// TwinCAT 3 PLC project Internship
// ProgramVersion: 3.1.4026.20
// libraries:
//   Tc2_Standard, * (Beckhoff Automation GmbH)
//   Tc2_System, * (Beckhoff Automation GmbH)
//   Tc3_Module, * (Beckhoff Automation GmbH)
// project tree:
//   Control/ FB_ControlSignal.TcPOU, FB_FeedForward.TcPOU, FB_FeedForward_NonLinear.TcPOU, FB_KvFF.TcPOU, FB_NaiveFF.TcPOU, FB_PID.TcPOU (not stored), FB_PressureFeedback.TcPOU, FB_Running.TcPOU (not stored), G_Mode.TcGVL (not stored)
//   Filtering/ FB_Filtering.TcPOU (not stored), G_Filtered.TcGVL (not stored)
//   GVL/ E_Mode.TcDUT (not stored), E_Motion.TcDUT, G_Enables.TcGVL, G_FilterConstants.TcGVL (not stored), G_OPC.TcGVL, G_Parameter.TcGVL
//   Inputs/Function Blocks/ FB_JoystickInputScaling.TcPOU, FB_Normalize.TcPOU (not stored), FB_PositionInputScaling.TcPOU
//   Inputs/ G_Inputs.TcGVL
//   MotionRef/ FB_AutoClock.TcPOU (not stored), FB_Home.TcPOU, FB_InitialPos.TcPOU (not stored), FB_MotionRef.TcPOU, FB_RunClock.TcPOU (not stored)
//   Outputs/ FB_ValveOutput.TcPOU (not stored), G_Output.TcGVL (not stored)
//   / PlcTask.TcTTO (not stored)
//   Programs/ MAIN.TcPOU (not stored), P_ControlBlock.TcPOU, P_FeedForward.TcPOU, P_Filtering.TcPOU (not stored), P_Inputs.TcPOU, P_Modes.TcPOU (not stored), P_Output.TcPOU, P_PID.TcPOU (not stored), P_RunClock.TcPOU (not stored)
//   XML/ FB_Derivator.TcPOU (not stored), G_Init.TcGVL (not stored), FB_Integrator.TcPOU (not stored)
// real-time tasks:
//   TASK PlcTask: cycle T#1ms, priority 20, ADS port 350
// I/O:
//   DEVICE Device 3 (EtherCAT), AmsNetId 192.168.0.204.4.1
//     RIO (EK1100) [EK1100 EtherCAT Coupler (2A E-Bus)]
//       DI (EL1008) [EL1008 8Ch. Dig. Input 24V, 3ms]
//       DO (EL2008) [EL2008 8Ch. Dig. Output 24V, 0.5A]
//       AI1 (EL3068) [EL3068 8Ch. Ana. Input 0-10V]
//       AI2 (EL3068) [EL3068 8Ch. Ana. Input 0-10V]
//       AI3 (EL3174) [EL3174 4Ch. Ana. Input +/-10V Diff., +/-20mA SingleEnded, 16 Bit]
//       AO (EL4104) [EL4104 4Ch. Ana. Output 0-10V, 16bit]
//       End Cap (EL9011) [EL9011 End Terminal]
// variable links:
//   Internship/Internship Instance <-> Device 3 (EtherCAT)/RIO (EK1100)/AI1 (EL3068)
//     PlcTask Inputs/G_Inputs.nRawJoystick <-> AI Standard Channel 2/Value
//     PlcTask Inputs/G_Inputs.nRawPistonPosition <-> AI Standard Channel 3/Value
//     PlcTask Inputs/G_Inputs.nRawSpoolPosition <-> AI Standard Channel 4/Value
//   Internship/Internship Instance <-> Device 3 (EtherCAT)/RIO (EK1100)/AI2 (EL3068)
//     PlcTask Inputs/G_Inputs.nRawPa <-> AI Standard Channel 4/Value
//     PlcTask Inputs/G_Inputs.nRawPaLower <-> AI Standard Channel 5/Value
//     PlcTask Inputs/G_Inputs.nRawPb <-> AI Standard Channel 6/Value
//     PlcTask Inputs/G_Inputs.nRawPs <-> AI Standard Channel 1/Value
//   Internship/Internship Instance <-> Device 3 (EtherCAT)/RIO (EK1100)/AI3 (EL3174)
//     PlcTask Inputs/G_Inputs.nRawFlowSensor <-> AI Standard Channel 1/Value
//   Internship/Internship Instance <-> Device 3 (EtherCAT)/RIO (EK1100)/AO (EL4104)
//     PlcTask Outputs/G_Output.nValveOutput <-> AO Output Channel 1/Analog output
//   Internship/Internship Instance <-> Device 3 (EtherCAT)/RIO (EK1100)/DI (EL1008)
//     PlcTask Inputs/G_Inputs.bAuto <-> Channel 1/Input
//     PlcTask Inputs/G_Inputs.bManual <-> Channel 2/Input
//     PlcTask Inputs/G_Inputs.bStartButton <-> Channel 3/Input
//     PlcTask Inputs/G_Inputs.bStopButton <-> Channel 4/Input
//   Internship/Internship Instance <-> Device 3 (EtherCAT)/RIO (EK1100)/DO (EL2008)
//     PlcTask Outputs/G_Output.bGreenLight <-> Channel 1/Output
//     PlcTask Outputs/G_Output.bRedLight <-> Channel 2/Output
//     PlcTask Outputs/G_Output.bRunning <-> Channel 3/Output

// ---- GVL/E_Motion.TcDUT
{attribute 'qualified_only'}
{attribute 'strict'}
{attribute 'to_string'}
TYPE E_Motion :
(
	Sine,
	Ramp
);
END_TYPE

// ---- GVL/G_Enables.TcGVL
{attribute 'qualified_only'}
VAR_GLOBAL
	
	// Control Enables
	bEnablePID 		: BOOL; // Enable PID Control
	bEnableFF 		: BOOL; // Enable FeedForward	
	bEnablePFB		: BOOL; // Enable Pressure Feedback
	bEnableU 		: BOOL; // Enable Signal to Valve

	bCharTesting	: BOOL; // Enable Characteristic testing
	bMove2Home		: BOOL; // Enable Home-function
	
	// No Function
	bEnableComp 	: BOOL; // Driving with Compensator
	

	// Enumerators
	nModeSelect		: E_Motion; // Motion Reference
	
END_VAR

// ---- GVL/G_OPC.TcGVL
{attribute 'qualified_only'}
VAR_GLOBAL
	
	// Unfiltered Pressures
	fPa 				: LREAL; // [bar], Pressure A 
	fPb 				: LREAL; // [bar], Pressure B 
	fPs 				: LREAL; // [bar], Pressure S 
	fPaLower 			: LREAL; // [bar], Pressure A inbetween DCV and CBV 
	
	// Filtered Pressures
	fPaFiltered 		: LREAL; // [bar], Pressure A Filtered 
	fPbFiltered 		: LREAL; // [bar], Pressure B Filtered
	fPsFiltered 		: LREAL; // [bar], Pressure S Filtered
	fPaLowerFiltered 	: LREAL; // [bar], Pressure A inbetween DCV and CBV Filtered
	
	fSpoolPosition 		: LREAL; // [-1..1], Spool position 
	fPistonPosition 	: LREAL; // [m], Piston position
	fPistonPosMeasured 	: LREAL; // [m], Measured piston position
	fJoystick 			: LREAL; // [-1..1], Joystick signal
	fFlow 				: LREAL; // [l/min], Flow rod side 
	fFlowCalc 			: LREAL; // [l/min], Calculated flow
	
	fXRef 				: LREAL; // [m], Position reference [m]
	fXDotRef 			: LREAL; // [m/s], Velocity reference [m/s]
	fFlowRef 			: LREAL; // [l/min], Flow reference calculated form fXDotRef
	
	fFFFlow				: LREAL; // [l/min], Flow form feed forward
	fKv					: LREAL;

	fWantedSpoolPos 	: LREAL; // [-1..1], Where spool is wanted to be
	fUpfbGrad 			: LREAL; // Pressure feedback gradient
	fPxGrad 			: LREAL; // Pressure gradient
	fUTest 				: LREAL; // [-1..1], Signal to Valve with pfb
	fTime 				: LREAL; // [s], Time
	fError 				: LREAL; // [m], Error
	
	
	fSignalPID 			: LREAL; // PID signal value
	fFF 				: LREAL; // FF signal Value
	fUpfb 				: LREAL; // Pressure feedback signal
	fU 					: LREAL; // [-1..1], Signal for spool to be where it is wanted


END_VAR

// ---- GVL/G_Parameter.TcGVL
{attribute 'qualified_only'}
VAR_GLOBAL
	// Motion Ref
	// Sine Parameters
	fAmplitude 		: LREAL := 0.15;
	fMean 			: LREAL := 0.2;
	fFrequency 		: LREAL := 0.05;
	
	
	// Valve Values
	// Flow
	fQMaxDown 		: LREAL := 10.0; // [L/min]
	fQMaxUp 		: LREAL := 10.0; // [L/min]	
	
	// Area
	fAreaUp 		: LREAL := 33.100/1E4; //[m^2]
	fAreaDown 		: LREAL := 23.560/1E4; //[m^2]
	
	// Deadband
	fDeadUp 		: LREAL := 0.23;
	fDeadDown 		: LREAL := 0.215;
	
	fMaxSpeed 		: LREAL := 0.01; // [m/s] 
	fDeltaP0 		: LREAL := 8.0; // [Bar]
	
	// Deadband test
	fConst 			: LREAL := 0.0; // [-1, 1]

	fCycleTime 		: LREAL := 0.001; // Time Step [s]
	fQConst 		: LREAL := 15;
	fPistonStroke 	: LREAL := 0.5;
	
	// PID-constants
	Kp 				: LREAL := 14.0; 	// P
	Ki 				: LREAL := 0.0;		// I
	Kd 				: LREAL := 0.0;		// D
	
	// Pressure feedback constants
	Kf				: LREAL := 2E-4;
	TauF			: LREAL := 0.1; // [0.05 .. 0.1]
	PFBstate		: INT 	:= 2; // 0:Switching, 1: Pa-phi*Pb, 2: Pb
	FFMode			: INT 	:= 1; // 0: Bachelor FF, 1: Kv FF, 2: Naive FF




END_VAR

// ---- Inputs/G_Inputs.TcGVL
{attribute 'qualified_only'}
VAR_GLOBAL
	// Mode Selector
	bManual 			AT %I* : BOOL;
	bAuto	 			AT %I* : BOOL;
	bStartButton		AT %I* : BOOL;
	bStopButton			AT %I* : BOOL;
	
	// Raw Pressure Values
	nRawPa 				AT %I*	: INT;
	nRawPb				AT %I*	: INT;
	nRawPs				AT %I*	: INT;
	nRawPaLower			AT %I* 	: INT;
	
	// Raw Position Values
	nRawPistonPosition 	AT %I*	: INT;
	nRawJoystick		AT %I*	: INT;
	nRawFlowSensor		AT %I*	: INT;
	nRawSpoolPosition	AT %I*	: INT;
END_VAR

// ---- Control/FB_ControlSignal.TcPOU
FUNCTION_BLOCK FB_ControlSignal
VAR_INPUT
	fFF 			: LREAL;
	fPID			: LREAL;
	fPFB			: LREAL;
	
	fDeadBandUp		: LREAL;
	fDeadBandDown	: LREAL;
	
	nFFState		: INT;

	bPID			: BOOL;
	bFF				: BOOL;
	bPFB			: BOOL;
	bU				: BOOL;
	bValve			: BOOL;
END_VAR
VAR_OUTPUT
	fU				: LREAL;
	fUAdj			: LREAL;
END_VAR
VAR
	FF				: LREAL;
	PID				: LREAL;
	PFB				: LREAL;
END_VAR


FF := fFF  * TO_INT(bFF);

PID := fPID * TO_INT(bPID);

PFB := fPFB * TO_INT(bPFB);

fUAdj := (FF+PID-PFB)*TO_INT(bValve);

IF FF = 0.0 THEN
	fU := 0.0;
ELSE
	CASE nFFState OF
		0: 
			IF (fUAdj > 0.0) THEN
				fU := fUAdj + fDeadBandUp;
			ELSIF (fUAdj < 0.0) THEN
				fU := fUAdj - fDeadBandDown;
			ELSE
				fU := 0.0;
			END_IF
			
		ELSE // FF States that use this: 1, 2
			IF (fUAdj > 0.0) THEN
				fU := fUAdj;
			ELSIF (fUAdj < 0.0) THEN
				fU := fUAdj;
			ELSE
				fU := 0.0;
			END_IF

		
	END_CASE
	
END_IF
IF fU < -1.0 THEN
	fU := -1.0;
ELSIF fU > 1.0 THEN
	fU := 1.0;
ELSE
	fU := fU;
END_IF

END_FUNCTION_BLOCK

// ---- Control/FB_FeedForward.TcPOU
FUNCTION_BLOCK FB_FeedForward
VAR_INPUT
	fXDotRef 		: LREAL; // Velocity Reference [m/s]
	fMaxFlowUp 		: LREAL; // Needs to be positive (22)
	fMaxFlowDown 	: LREAL; // Needs to be positive (15)
	fDeadUp			: LREAL; // Needs to be positive (0.155)
	fDeadDown 		: LREAL; // Needs to be positive (0.18)

	fPs 			: LREAL; // [Bar]
	fPa 			: LREAL; // [Bar]
	fPb 			: LREAL; // [Bar]
	fDeltaP0		: LREAL; // [Bar]
	fAreaUp			: LREAL; // [mm^2]
	fAreaDown		: LREAL; // [mm^2]

END_VAR
VAR_OUTPUT
	fUFF 			: LREAL;
	fFlow			: LREAL; 	// Wanted Flow
	fFlowLM			: LREAL;	// Flow [L/min]
END_VAR
VAR

	fDeltaP_Norm	: LREAL; 	// Pressure Drop with Compansator
	
	fDeltaP			: LREAL; 	// Pressure Drop
	fDeltaP_Ref		: LREAL; 	// Referance Pressure Drop
	fFlowRef		: LREAL; 	// Refereance Flow
	
	fUFFTemp		: LREAL;	// Temp Signal Out
END_VAR


fDeltaP_Norm	:= fDeltaP0 * 100000.0;

IF fXDotRef > 0.0 THEN
	
	fFlow := fXDotRef * fAreaUp;
	fFlowLM := -fFlow * 60000;
	fDeltaP := (fPs - fPa) * 100000.0;
	IF fDeltaP < 100 THEN
		fDeltaP := 100;
	ELSE
		fDeltaP := fDeltaP;
	END_IF
	fDeltaP_Ref := ABS(fDeltaP_Norm/ (fDeltaP));
	fFlowRef := (fFlow * SQRT(fDeltaP_Ref)) * 60000.0;
	fUFFTemp := fFlowRef/fMaxFlowUp;
	fUFFTemp := -fUFFTemp * (1.0-fDeadUp);
	
ELSIF fXDotRef < 0.0 THEN
	
	fFlow := fXDotRef * fAreaDown;
	fFlowLM := -fFlow * 60000;
	fDeltaP := (fPs - fPb) * 100000.0;
	IF fDeltaP < 100 THEN
		fDeltaP := 100;
	ELSE
		fDeltaP := fDeltaP;
	END_IF
	fDeltaP_Ref := ABS(fDeltaP_Norm/(fDeltaP));
	fFlowRef := (fFlow * SQRT(fDeltaP_Ref)) * 60000.0;
	fUFFTemp := fFlowRef/fMaxFlowDown; 
	fUFFTemp := -fUFFTemp*(1.0-fDeadDown);
	
ELSE
	
	fUFFTemp := 0.0;		

END_IF

IF fUFFTemp > 1.0 THEN
	fUFF := 1.0;
ELSIF fUFFTemp < -1.0 THEN
	fUFF := -1.0;
ELSE
	fUFF := fUFFTemp;
END_IF

END_FUNCTION_BLOCK

// ---- Control/FB_FeedForward_NonLinear.TcPOU
FUNCTION_BLOCK FB_FeedForward_NonLinear
VAR_INPUT
	fXDotRef 		: LREAL; // Velocity Reference [m/s]
	fMaxFlowUp 		: LREAL; // Needs to be positive (22)
	fMaxFlowDown 	: LREAL; // Needs to be positive (15)
	fDeadUp			: LREAL; // Needs to be positive (0.155)
	fDeadDown 		: LREAL; // Needs to be positive (0.18)

	fPs 			: LREAL; // [Bar]
	fPa 			: LREAL; // [Bar]
	fPb 			: LREAL; // [Bar]
	fDeltaP0		: LREAL; // [Bar]
	fAreaUp			: LREAL; // [mm^2]
	fAreaDown		: LREAL; // [mm^2]

END_VAR
VAR_OUTPUT
	fUFF 			: LREAL;
	fFlow			: LREAL; 	// Wanted Flow
	fFlowLM			: LREAL;	// Flow [L/min]
END_VAR
VAR

	fDeltaP_Norm	: LREAL; 	// Pressure Drop with Compansator
	
	fDeltaP			: LREAL; 	// Pressure Drop
	fDeltaP_Ref		: LREAL; 	// Referance Pressure Drop
	fFlowRef		: LREAL; 	// Refereance Flow
	
	fUFFTemp		: LREAL;	// Temp Signal Out
END_VAR


fDeltaP_Norm	:= fDeltaP0 * 100000.0;

IF fXDotRef > 0.0 THEN
	
	fFlow := fXDotRef * fAreaUp;
	fFlowLM := -fFlow * 60000;
	fDeltaP := (fPs - fPa) * 100000.0;
	IF fDeltaP < 100 THEN
		fDeltaP := 100;
	ELSE
		fDeltaP := fDeltaP;
	END_IF
	fDeltaP_Ref := ABS(fDeltaP_Norm/ (fDeltaP));
	fFlowRef := (fFlow * SQRT(fDeltaP_Ref)) * 60000.0;
	fUFFTemp := fFlowRef/fMaxFlowUp;
	fUFFTemp := -fUFFTemp * (1.0-fDeadUp);
	
ELSIF fXDotRef < 0.0 THEN
	
	fFlow := fXDotRef * fAreaDown;
	fFlowLM := -fFlow * 60000;
	fDeltaP := (fPs - fPb) * 100000.0;
	IF fDeltaP < 100 THEN
		fDeltaP := 100;
	ELSE
		fDeltaP := fDeltaP;
	END_IF
	fDeltaP_Ref := ABS(fDeltaP_Norm/(fDeltaP));
	fFlowRef := (fFlow * SQRT(fDeltaP_Ref)) * 60000.0;
	fUFFTemp := fFlowRef/fMaxFlowDown; 
	fUFFTemp := -fUFFTemp*(1.0-fDeadDown);
	
ELSE
	
	fUFFTemp := 0.0;		

END_IF

IF fUFFTemp > 1.0 THEN
	fUFF := 1.0;
ELSIF fUFFTemp < -1.0 THEN
	fUFF := -1.0;
ELSE
	fUFF := fUFFTemp;
END_IF

END_FUNCTION_BLOCK

// ---- Control/FB_KvFF.TcPOU
FUNCTION_BLOCK FB_KvFF
VAR_INPUT
	fPs 		: LREAL; // [bar]
	fPa 		: LREAL; // [bar]
	fPb 		: LREAL; // [bar]
	
	fXDotRef 	: LREAL; // [m/s]
END_VAR
VAR_OUTPUT
	fFFTemp		: LREAL; // [-1..1], Wanted spool position, u
	fFF 		: LREAL; // [-1..1], Spool signal for position, ~u
	fFlow 		: LREAL; // [l/min]
	fKv 		: LREAL; // [l/min / bar^0.5]
END_VAR
VAR
	fDeltaP		: LREAL; // [bar]
END_VAR




IF fXDotRef > 0.0 THEN
	IF fKv >= 0.1 THEN
		fFFTemp := -0.013*EXPT(fKv,5) + 0.1355*EXPT(fKv,4) - 0.5012*EXPT(fKv,3) + 0.7175*EXPT(fKv,2) - 0.0278 * fKv + 0.2684;
	ELSIF fKv < 0.1 THEN
		fFFTemp := 0.2325 + 0.0398 * fKv/0.1;
	ELSE 
		fFFTemp := G_Parameter.fDeadUp;
	END_IF
	fFlow := fXDotRef * G_Parameter.fAreaUp * 6E4;
	fDeltaP := fPs - fPa;
	
	fFF := -(fFFTemp + 0.0151)/1.1224;
ELSIF fXDotRef < 0.0 THEN
	IF fKv >= 0.1 THEN
		fFFTemp := 0.0054*EXPT(fKv,6) - 0.0733*EXPT(fKv,5) + 0.3796*EXPT(fKv,4) - 0.9356*EXPT(fKv,3) + 1.0359*EXPT(fKv,2) - 0.1046 * fKv + 0.2381;
	ELSIF fKv < 0.1 THEN
		fFFTemp := 0.2175 + 0.0196 * fKv/0.1;
	ELSE 
		fFFTemp := G_Parameter.fDeadDown;
	END_IF
	fFlow := fXDotRef * G_Parameter.fAreaDown * 6E4;
	fDeltaP := fPs - fPb;
	fFF := (fFFTemp + 0.0398)/1.1079;
ELSE
	fFlow := 0.0;
	fFFTemp := 0.0;
	fFF := 0.0;
END_IF

IF fDeltaP <= 0.0 THEN
	fKv := 4.0;
ELSE
	fKv := ABS(fFlow)/SQRT(fDeltaP);
END_IF

END_FUNCTION_BLOCK

// ---- Control/FB_NaiveFF.TcPOU
FUNCTION_BLOCK FB_NaiveFF
VAR_INPUT
	fPs 		: LREAL; // [bar]
	fPa 		: LREAL; // [bar]
	fPb 		: LREAL; // [bar]
	
	fXDotRef 	: LREAL; // [m/s]
END_VAR
VAR_OUTPUT

	fFF 		: LREAL; // [-1..1], Spool signal for position, u
	fFlow 		: LREAL; // [l/min]
	fKv 		: LREAL; // [l/min / bar^0.5]
END_VAR
VAR
	fDeltaP		: LREAL; // [bar]
END_VAR




IF fXDotRef > 0.0 THEN
	fFlow := fXDotRef * G_Parameter.fAreaUp * 6E4;
	fDeltaP := fPs - fPa;
	
	fFF := -(0.2143 + 0.7857 * fKv/3.7796);
ELSIF fXDotRef < 0.0 THEN
	fFlow := fXDotRef * G_Parameter.fAreaDown * 6E4;
	fDeltaP := fPs - fPb;
	
	fFF := (0.2143 + 0.7857 * fKv/3.7796);
ELSE
	fFlow := 0.0;
	fFF := 0.0;
END_IF

IF fDeltaP <= 0.0 THEN
	fKv := 4.0;
ELSE
	fKv := ABS(fFlow)/SQRT(fDeltaP);
END_IF

END_FUNCTION_BLOCK

// ---- Control/FB_PressureFeedback.TcPOU
FUNCTION_BLOCK FB_PressureFeedback
VAR_INPUT
	fKf			: LREAL;
	fTauF		: LREAL; // [s]	
	state		: INT;
END_VAR
VAR_OUTPUT
	fUpfb 		: LREAL;
	fUpfbGrad	: LREAL;
	fPxGrad		: LREAL; // [Bar]
END_VAR
VAR
	fDt			: LREAL := 0.001; // [s]
	fPx			: LREAL := 0.0; // [Bar]
	fPxOld		: LREAL; // [Bar]
	fARatio		: LREAL;
END_VAR


CASE state OF
	0: // Altering input for Px
		IF G_OPC.fU < 0.0 THEN
			fPx := G_OPC.fPa;
		ELSIF G_OPC.fU > 0.0 THEN
			fPx := G_OPC.fPb;
		ELSE
			fPx := 0.0;
		END_IF
	1:	// Px = Pa - phi * Pb
		fARatio := G_Parameter.fAreaDown/G_Parameter.fAreaUp;
		fPx := G_OPC.fPa - fARatio * G_OPC.fPb;
	2:	// Px = Pb
		fPx := G_OPC.fPb;
END_CASE

fPxGrad := (fPx - fPxOld)/fDt;
fUpfbGrad :=  (fKf * fPxGrad - fUpfb)/fTauF;
fUpfb := fUpfb + fUpfbGrad * fDt;

fPxOld := fPx;

END_FUNCTION_BLOCK

// ---- Inputs/Function Blocks/FB_JoystickInputScaling.TcPOU
FUNCTION_BLOCK FB_JoystickInputScaling
VAR_INPUT
	bEnable 				: BOOL;
	nRawInput 				: INT;
	fMaxValue 				: LREAL;
	fMaxInputValue			: LREAL;
	fMinInputValue 			: LREAL;
	fNeutralInputValue  	: LREAL;
	fNeutralDeadband		: LREAL;
END_VAR
VAR_OUTPUT
	fOutput : LREAL;
END_VAR
VAR
	fRawInput : LREAL;
	fTempInput : LREAL;
	fTempOutput : LREAL;

	fMaxOutputValue  		: LREAL := 1.0;
	fMinOutputValue  		: LREAL := -1.0;
	fNeutralOutputValue  	: LREAL := 0.0;
END_VAR

fRawInput := INT_TO_LREAL(nRawInput);

fTempInput := fRawInput - fNeutralInputValue;

IF fTempInput > fNeutralDeadband THEN
	fTempOutput := fTempInput/(fMaxInputValue - fNeutralInputValue);
ELSIF fTempInput < -fNeutralDeadband THEN	
	fTempOutput := fTempInput/(fNeutralInputValue - fMinInputValue);
ELSE
	fTempOutput := 0.0;
END_IF

IF NOT(bEnable) THEN
	fOutput := 0.0;
ELSE
	fOutput := LIMIT(fMinOutputValue * fMaxValue, fTempOutput * fMaxValue, fMaxOutputValue* fMaxValue);
END_IF

END_FUNCTION_BLOCK

// ---- Inputs/Function Blocks/FB_PositionInputScaling.TcPOU
FUNCTION_BLOCK FB_PositionInputScaling
VAR_INPUT
	nRawInput 				: INT;
	fMaxInputValue 			: LREAL;
	fMinInputValue			: LREAL;
	fMaxOutputValue  		: LREAL;
	fMinOutputValue  		: LREAL;	
END_VAR
VAR_OUTPUT
	fOutput : LREAL;
	fActual : LREAL;
END_VAR
VAR
	fRawInput : LREAL;
	fNormalizedInput: LREAL;
	fTempOut : LREAL;
END_VAR

fRawInput := INT_TO_LREAL(nRawInput);

fNormalizedInput := (fRawInput - fMinInputValue) / (fMaxInputValue - fMinInputValue);
fTempOut := fMinOutputValue + fNormalizedInput*(fMaxOutputValue - fMinOutputValue);

fOutput := LIMIT(fMinOutputValue, fTempOut, fMaxOutputValue);
fActual := LIMIT(fMinOutputValue, fTempOut - 0.0006 - 0.0109*fTempOut + 0.5855*EXPT(fTempOut,2) - 1.1291*EXPT(fTempOut,3), fMaxOutputValue);

END_FUNCTION_BLOCK

// ---- MotionRef/FB_Home.TcPOU
FUNCTION_BLOCK FB_Home
VAR_INPUT
	bGoHome : BOOL;
	fCurrentPos : LREAL; // [m]
	fTolerance : LREAL; // [m]
	fMoveTime : LREAL; // [s]
	fHomePos : LREAL; // [m]
	fMoveTimer : LREAL; // [s]
END_VAR
VAR_OUTPUT
	fXRef : LREAL; // [m]
	fXDotRef : LREAL; // [m/s]
END_VAR
VAR
	
END_VAR




IF bGoHome AND ABS(fHomePos-fCurrentPos)>fTolerance THEN
	fXDotRef := (fHomePos-fCurrentPos)/fMoveTime;
	fXRef := fCurrentPos + fXDotRef * fMoveTimer;
	IF	ABS(fHomePos-fCurrentPos)<=fTolerance THEN
		bGoHome := FALSE;
		fXDotRef := 0.0;
		fXRef := fCurrentPos;
	END_IF
ELSE
	fXDotRef := 0.0;
	fXRef := fCurrentPos;
END_IF

END_FUNCTION_BLOCK

// ---- MotionRef/FB_MotionRef.TcPOU
FUNCTION_BLOCK FB_MotionRef
VAR_INPUT
	fAmplitude : LREAL;
	fFrequency : LREAL;
	fInitialPos : LREAL;
	fCurrentPos : LREAL;
	nMotionMode : INT;
	fMotionTimer 	: LREAL;           // For selve rampen
END_VAR
VAR_OUTPUT
	fXDotRef : LREAL;
	fXRef : LREAL;
	fWantedFlow : LREAL;
END_VAR
VAR
	fPI : LREAL := 3.1415;
	fMean : LREAL;
	
	arrBounduary 	: ARRAY[0..1] OF LREAL := [G_Parameter.fPistonStroke * 0.1, G_Parameter.fPistonStroke * 0.9]; // Min, Max [m]
	fRampTime 	 	: LREAL := 15.0; // [s]
 	fTolerance   	: REAL := 0.005;  // ±5 mm
  	
END_VAR




CASE nMotionMode OF
	0:	// Sine
	
		fMean := fAmplitude + fInitialPos; 
		fXRef := fMean - fAmplitude * COS(2*fPI * fFrequency * fMotionTimer);
		fXDotRef := 2 * fPI *fFrequency * fAmplitude * SIN(2*fPI * fFrequency * fMotionTimer); 
		
	1:	// Ramp


		IF fMotionTimer <= fRampTime THEN
			fXDotRef := (arrBounduary[1] - arrBounduary[0]) / fRampTime;
			fXRef := arrBounduary[0] + fXDotRef * fMotionTimer;
		ELSIF fMotionTimer <= fRampTime * (4.0/3.0) THEN
			fXRef := arrBounduary[1];
			fXDotRef := 0.0;
		ELSIF fMotionTimer <= (2.0 + 1.0/3.0) * fRampTime AND fMotionTimer > fRampTime * (4.0/3.0) THEN
			fXDotRef := (arrBounduary[0] - arrBounduary[1]) / fRampTime;
			fXRef := arrBounduary[1] + fXDotRef * (fMotionTimer - (4.0/3.0) * fRampTime);
		ELSIF fMotionTimer > (2.0 + 1.0/3.0) * fRampTime THEN
			fXDotRef := 0.0;
			fXRef := arrBounduary[0];
		END_IF
END_CASE

IF fXDotRef > 0.0 THEN
	fWantedFlow := fXDotRef * G_Parameter.fAreaUp*6E4;
ELSIF fXDotRef < 0.0 THEN
	fWantedFlow := fXDotRef * G_Parameter.fAreaDown*6E4;
ELSE
	fWantedFlow := 0.0;
END_IF

END_FUNCTION_BLOCK

// ---- Programs/P_ControlBlock.TcPOU
PROGRAM P_ControlBlock
VAR
	fbAutoClock : FB_AutoClock;
	fbMotionRef : FB_MotionRef;
	fbControl : FB_ControlSignal;
	fbInitialPos : FB_InitialPos;
	nMode : E_Motion;
	fbPressureFB : FB_PressureFeedback;
	fbHome : FB_Home;
	StartTimer : TON;
END_VAR


fbControl(
	nFFState := G_Parameter.FFMode,	

	bFF := G_Enables.bEnableFF,
	bPID := G_Enables.bEnablePID,
	bPFB := G_Enables.bEnablePFB,
	bU := G_Enables.bEnableU,
	bValve := TRUE,
	
	fDeadBandUp := G_Parameter.fDeadUp,
	fDeadBandDown := G_Parameter.fDeadDown
);

fbPressureFB(
			fKf := G_Parameter.Kf,
			fTauF := G_Parameter.TauF,
			state := G_Parameter.PFBstate,
			
			fUpfb => G_OPC.fUpfb,
			fUpfbGrad => G_OPC.fUpfbGrad,
			fPxGrad => G_OPC.fPxGrad
		);

IF G_Mode.bAuto AND G_Mode.bRunning THEN

	fbInitialPos(
		bEnable := G_Inputs.bStartButton,
		fCurrentPos := G_OPC.fPistonPosition
	);
	
	fbAutoClock(
		fStart := StartTimer.Q,
		fRunning := G_Mode.bRunning,
		fCycle := G_Parameter.fCycleTime
	);
	
	IF G_Inputs.bStartButton THEN
		StartTimer(IN := TRUE, PT :=T#2S);
		fbMotionRef();
		IF StartTimer.Q THEN
			
			IF G_Enables.bMove2Home THEN 
				fbHome(
					bGoHome := G_Enables.bMove2Home,
					fCurrentPos := G_OPC.fPistonPosition,
					fHomePos := 0.05,
					fMoveTimer := fbAutoClock.fTime,
					fMoveTime := 10.0,
					fTolerance := 0.002,
					
					fXDotRef => G_OPC.fXDotRef,
					fXRef => G_OPC.fXRef
				);
			ELSE
			fbMotionRef(
				nMotionMode := G_Enables.nModeSelect,
				fMotionTimer := fbAutoClock.fTime,
				fAmplitude := G_Parameter.fAmplitude,
				fInitialPos := fbInitialPos.fInitialPos,
				fFrequency := G_Parameter.fFrequency,
				fCurrentPos := G_OPC.fPistonPosition,
				fXDotRef => G_OPC.fXDotRef,
				fXRef => G_OPC.fXRef,
				fWantedFlow => G_OPC.fFlowRef
			);
			END_IF
		ELSE 
			G_OPC.fXDotRef := 0.0;
			G_OPC.fXRef := G_OPC.fPistonPosition;
		END_IF
	ELSE 
		StartTimer(IN := FALSE);
		G_OPC.fXDotRef := 0.0;
		G_OPC.fXRef := G_OPC.fPistonPosition;
	END_IF
	
	
	G_OPC.fUTest := G_OPC.fU - G_OPC.fUpfb;
	
	fbControl(
		fFF := G_OPC.fFF,
		fPID := G_OPC.fSignalPID,
		fPFB := G_OPC.fUpfb,
		
		fU => G_OPC.fU
	);
		
		
	
	

ELSIF G_Mode.bManual AND G_Mode.bRunning THEN

	fbInitialPos(
		bEnable := G_Inputs.bStartButton,
		fCurrentPos := G_OPC.fPistonPosition
	);
	
	IF G_Enables.bCharTesting THEN
		IF G_OPC.fPistonPosition >= 0.9*0.5 OR G_OPC.fPistonPosition <= 0.1 * 0.5 THEN
			G_OPC.fU := 0.0;
		ELSE
			G_OPC.fU := G_Parameter.fConst - G_OPC.fUpfb * TO_INT(G_Enables.bEnablePFB);
		END_IF
	
	ELSE
		G_OPC.fU := G_OPC.fJoystick;
	END_IF
	
END_IF

END_PROGRAM

// ---- Programs/P_FeedForward.TcPOU
PROGRAM P_FeedForward
VAR
	fbFF 	: FB_FeedForward;
	fbKv 	: FB_KvFF;
	fbNaive	: FB_NaiveFF;
END_VAR

//fbKv(
//	fPa := G_OPC.fPa,
//	fPb := G_OPC.fPb,
//	fPs := G_OPC.fPs,
	
//	fXDotRef := G_OPC.fXDotRef,
	
//	fUTemp => G_OPC.fWantedSpoolPos,
//	fU => G_OPC.fU
//);

	
CASE G_Parameter.FFMode OF
	0:
		fbFF(
			fMaxFlowUp := G_Parameter.fQMaxUp,
			fMaxFlowDown := G_Parameter.fQMaxDown,
			fDeadUp := G_Parameter.fDeadUp,
			fDeadDown := G_Parameter.fDeadDown,
			fAreaUp := G_Parameter.fAreaUp,
			fAreaDown := G_Parameter.fAreaDown,
			
			fPs := G_OPC.fPs,
			fPa := G_OPC.fPa,
			fPb := G_OPC.fPb,
			fDeltaP0 := G_Parameter.fDeltaP0,
			
			fXDotRef := G_OPC.fXDotRef,		
	
			fUFF => G_OPC.fFF,
			fFlowLM => G_OPC.fFlowCalc
		);
		
	1:
		fbKv(
			fPa :=G_OPC.fPaLower,
			fPb := G_OPC.fPb,
			fPs := G_OPC.fPs,
			
			fXDotRef := G_OPC.fXDotRef,
			
			fFFTemp => G_OPC.fWantedSpoolPos,
			fFF => G_OPC.fFF,
			fFlow => G_OPC.fFFFlow,
			fKv => G_OPC.fKv
			
			
		);
	2:
		fbNaive(
			fPa :=G_OPC.fPaLower,
			fPb := G_OPC.fPb,
			fPs := G_OPC.fPs,
			
			fXDotRef := G_OPC.fXDotRef,
			
			fFF => G_OPC.fFF,
			fFlow => G_OPC.fFFFlow,
			fKv => G_OPC.fKv
		);
		

END_CASE

END_PROGRAM

// ---- Programs/P_Inputs.TcPOU
PROGRAM P_Inputs
VAR
	fbNormPa :  FB_Normalize;
	fbNormPb :  FB_Normalize;
	fbNormPs :  FB_Normalize;
	fbNormPaLower : FB_Normalize;
	
	fbNormPistonPosition : FB_PositionInputScaling;
	fbNormSpoolPosition : FB_JoystickInputScaling;
	fbJoystick : FB_JoystickInputScaling;
	fbFlow	: FB_JoystickInputScaling;

	fPa : LREAL;
	fPb : LREAL;
	fPs : LREAL;
	fPaLower : LREAL;
	
	fPistonPosition : LREAL;
END_VAR

fbNormPa(
	nRawInput := G_Inputs.nRawPa,
	fMaxValue := 400.0, 			// [Bar]
	fNormalizedInput => G_OPC.fPa
);

fbNormPb(
	nRawInput := G_Inputs.nRawPb,
	fMaxValue := 400.0, 			// [Bar]
	fNormalizedInput => G_OPC.fPb
);

fbNormPs(
	nRawInput := G_Inputs.nRawPs,
	fMaxValue := 400.0, 			// [Bar]
	fNormalizedInput => G_OPC.fPs
);

fbNormPistonPosition(
	nRawInput := G_Inputs.nRawPistonPosition,
	
	fMaxInputValue := 16090.0,
	fMinInputValue := 125.0,
	fMaxOutputValue := 0.5,
	fMinOutputValue := 0.0,	
	
	fOutput => G_OPC.fPistonPosMeasured,
	fActual => G_OPC.fPistonPosition
);
	
fbJoystick(
	nRawInput := G_Inputs.nRawJoystick,
	fMaxValue := 1.0,
	bEnable := (G_Mode.bRunning AND G_Mode.bManual),
	
	fMaxInputValue := 14746.0,
	fMinInputValue := 1617.0,
	fNeutralInputValue := 8160.0,
	fNeutralDeadband := 100.0,
	
	fOutput => G_OPC.fJoystick
);

fbNormPaLower(
	nRawInput := G_Inputs.nRawPaLower,
	fMaxValue := 400.0, 			// [Bar]
	fNormalizedInput => G_OPC.fPaLower
);

fbNormSpoolPosition(
	nRawInput := G_Inputs.nRawSpoolPosition,
	fMaxValue := 1.0,
	bEnable := TRUE,
	
	fNeutralInputValue := 8355.0,
	fMaxInputValue := 12645.0,
	fMinInputValue := 4071,
	fNeutralDeadband := 15.0,
	
	fOutput => G_OPC.fSpoolPosition
);

fbFlow(
	bEnable := TRUE,
	nRawInput := G_Inputs.nRawFlowSensor,
	fMaxValue := 150.0, // [l/min]
	
	fMaxInputValue := 32767.0,
	fMinInputValue := 0,
	fNeutralInputValue := 15270.0,
	fNeutralDeadband := 25.0,
	
	fOutput => G_OPC.fFlow
);

END_PROGRAM

// ---- Programs/P_Output.TcPOU
PROGRAM P_Output
VAR
	fbValveOutput : FB_ValveOutput;
END_VAR


fbValveOutput(
	fNormalizedInput := G_OPC.fU,
	bEnable := G_Enables.bEnableU,
	nOutput => G_Output.nValveOutput	
);

IF G_Mode.bRunning THEN
	G_Output.bGreenLight := TRUE;
	G_Output.bRedLight := TRUE;
ELSE
	G_Output.bGreenLight := FALSE;
	G_Output.bRedLight := FALSE;
END_IF

END_PROGRAM
